Yaskawa INFORM job: BABY.JBI

/JOB
//NAME BABY
//POS
///NPOS 7,0,0,0
///TOOL 0
///RECTAN
C000=0.000,0.000,0.000,0.000,0.000,0.000
C001=0.000,0.000,0.000,0.000,0.000,0.000
C002=0.000,0.000,0.000,0.000,0.000,0.000
C003=0.000,0.000,0.000,0.000,0.000,0.000
C004=0.000,0.000,0.000,0.000,0.000,0.000
C005=0.000,0.000,0.000,0.000,0.000,0.000
C006=0.000,0.000,0.000,0.000,0.000,0.000
//INST
///DATE 2014/09/13 22:59
///ATTR 0,0,0,0,0,0,0,0,0,0,0,0,1,1,0,0
///FRAME BASE
NOP
END
